{attribute 'qualified_only'}
VAR_GLOBAL
END_VAR

(* stored: Version 1.1.0.1, ProductVersion 3.1.4024.12
   GVL M001: Id {765ee5e2-ad3e-0896-2729-bcc1475f9821} *)
